// Mitsubishi GX Works2 project: CC-link_B_register   PLC: Q03UDV

PROGRAM MAIN
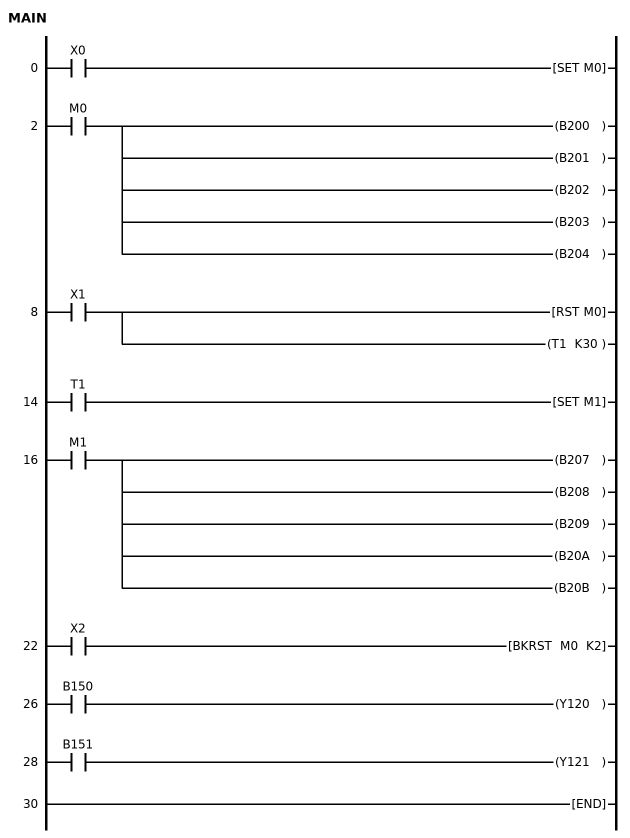
0     LD      X0
      SET     M0
2     LD      M0
      OUT     B200
      OUT     B201
      OUT     B202
      OUT     B203
      OUT     B204
8     LD      X1
      RST     M0
      OUT     T1 K30
14    LD      T1
      SET     M1
16    LD      M1
      OUT     B207
      OUT     B208
      OUT     B209
      OUT     B20A
      OUT     B20B
22    LD      X2
      BKRST   M0 K2
26    LD      B150
      OUT     Y120
28    LD      B151
      OUT     Y121
30    END
END_PROGRAM
